TYPE "PosList_IAI"
VERSION : 0.1
   STRUCT
      List : Array[0..39] of Struct
         Pos : Real;
         Vel : Int;
      END_STRUCT;
   END_STRUCT;

END_TYPE

